(* CoDeSys 2.3 export: PLC_TO_SCADA.EXP *)

(* POU PRG/PLC_TO_SCADA, ST *)
PROGRAM PLC_TO_SCADA
VAR
END_VAR
;
END_PROGRAM
